Fanuc KAREL source: kx00018.KL

-- PROVISIONAL review KL for V1013-1; original PC SHA256 c08e30b699ab671d74abb203ae916d8e5202969f1616244dd7eeeddeebed55cc
-- Incomplete behavior may be omitted. Consult companion uncertainty JSON. Do not deploy.
PROGRAM KX00018
%NOLOCKGROUP
VAR
  I : INTEGER
  J : INTEGER
  B : BOOLEAN
  F : FILE
  S : STRING[80]
-- UNRESOLVED_DECL P type=000102
-- UNRESOLVED_DECL BA type=002018
BEGIN
  -- UNRESOLVED_PC offsets 5-19; opcodes 2E,22,9D,33,B2
  -- UNRESOLVED_PC offsets 24-39; opcodes 22,9D,33,B1,23
  -- UNRESOLVED_PC offsets 44-48; opcodes 7F
END KX00018
